// TIA Portal V18 export
// export: Created 2025-12-01T12:38:41.2842192Z, ExportSetting None, DisplayName Totally Integrated Automation Portal, DisplayVersion V18 Update 5, DisplayName TIA Portal Openness, DisplayVersion V18 Update 5, DisplayName TIA Portal Teamcenter Gateway, DisplayVersion V18, DisplayName TIA Portal Version Control Interface, DisplayVersion V18, DisplayName STEP 7 Professional, DisplayVersion V18 Update 5, DisplayName STEP 7 Safety, DisplayVersion V18, DisplayName WinCC Professional, DisplayVersion V18 Update 5
DATA_BLOCK "KistlerPressData2"   // DB2321
{ S7_Optimized_Access := 'FALSE' }
// stored: AutoNumber false
   VAR
      Spare : Struct
         Spare : Array[0..85] of Byte;
      END_STRUCT;
      Data : Struct
         EO01 : Struct
            "pvXMin-Y" : Real;
            "pvXMax-Y" : Real;
            "pvXMin-X" : Real;
            "pvXMax-X" : Real;
         END_STRUCT;
         EO02 : Struct
            "pvXMin-Y" : Real;
            "pvXMax-Y" : Real;
            "pvXMin-X" : Real;
            "pvXMax-X" : Real;
         END_STRUCT;
         EO03 : Struct
            "pvXMax-Y" : Real;
            "pvXMax-X" : Real;
         END_STRUCT;
      END_STRUCT;
      iWritePressData : Struct
         temp1 : Real;
      END_STRUCT;
      PressData1 : Struct
         pvBlock_X : Real;
         pvBlock_Y : Real;
      END_STRUCT;
      ManualPro : Int;
   END_VAR
BEGIN
END_DATA_BLOCK
